(* Logix 5000 project; controller HP_SSC01hv vendor 1 type 14 code 158 rev 32.11; software revision 32.03; part 7 of 15 *)
(* tags used below, declared in another part *)
   A_C2_0422 : ALIAS FOR C2_Warning.22;
   A_C2_0423 : ALIAS FOR C2_Warning.23;
   A_C2_0425 : ALIAS FOR C2_Warning.25;
   A_C2_0426 : ALIAS FOR C2_Warning.26;
   C1_MAG : MOTION_INSTRUCTION;
   C1_MAS : MOTION_INSTRUCTION;
   C2_32HourTimers : TIMER[4];
   C2_ActualPositionMOD60 : REAL;
   C2_All_DLY_OK : BOOL;
   C2_Brake_Daily_ok : BOOL;
   C2_BrakeReleaseSelected : BOOL;
   C2_BrakeTestExpireTime : DINT;
   C2_BrakeTestExpireTimeTemp : DINT;
   C2_BrakeTestFailed : BOOL;
   C2_BrakeTestMessageNumber : DINT;
   C2_BrakeTestSelected : BOOL;
   C2_BrakeTestSequence : DINT;
   C2_BrakeTestWarning : BOOL;
   C2_DistanceToEvac : REAL;
   C2_Dump_OK : BOOL;
   C2_DumpValveReleaseSelected : BOOL;
   C2_DumpValveTestExpireTime : DINT;
   C2_DumpValveTestExpireTimeTemp : DINT;
   C2_DumpValveTestSelected : BOOL;
   C2_DumpValveTestSequence : DINT;
   C2_EvacPosition : REAL;
   C2_EvacPositionMOD60 : REAL;
   C2_ExcecutePBHoldTimer : TIMER;
   C2_FaultStandard : DINT;
   C2_GoNearOnPathDelay : TIMER;
   C2_GoToEvacMAM01 : MOTION_INSTRUCTION;
   C2_GoToOnPathMAM01 : MOTION_INSTRUCTION;
   C2_GoToOnPathMAM02 : MOTION_INSTRUCTION;
   C2_Home_OK : BOOL;
   C2_Homed : BOOL;
   C2_HomeExpireTime : DINT;
   C2_HomeExpireTimeTemp : DINT;
   C2_HomeSequence : DINT;
   C2_JogForwardFastSelected : BOOL;
   C2_JogForwardSlowSelected : BOOL;
   C2_JogReverseFastSelected : BOOL;
   C2_JogReverseSlowSelected : BOOL;
   C2_LubricationMessageNumber : DINT;
   C2_LubricationOnTimer : TIMER;
   C2_LubricationOverrideSelected : BOOL;
   C2_MAFR : MOTION_INSTRUCTION;
   C2_MAJDeceleration : REAL;
   C2_MASR : MOTION_INSTRUCTION;
   C2_Oiler : ALIAS FOR C2_RIO_AENT:O.Data[2].1;
   C2_OIT_BrakeRelease : BOOL;
   C2_OIT_BrakeReleaseDisplay : BOOL;
   C2_OIT_BrakeTest : BOOL;
   C2_OIT_BrakeTestDisplay : BOOL;
   C2_OIT_Command : DINT;
   C2_OIT_Current : DINT;
   C2_OIT_DumpValveRelease : BOOL;
   C2_OIT_DumpValveReleaseDisplay : BOOL;
   C2_OIT_DumpValveTest : BOOL;
   C2_OIT_DumpValveTestDisplay : BOOL;
   C2_OIT_FaultsExist : BOOL;
   C2_OIT_HomeCountDown : DINT;
   C2_OIT_JogForwardFast : BOOL;
   C2_OIT_JogForwardFastDisplay : BOOL;
   C2_OIT_JogForwardSlow : BOOL;
   C2_OIT_JogForwardSlowDisplay : BOOL;
   C2_OIT_JogReverseFast : BOOL;
   C2_OIT_JogReverseFastDisplay : BOOL;
   C2_OIT_JogReverseSlow : BOOL;
   C2_OIT_JogReverseSlowDisplay : BOOL;
   C2_OIT_JogStopDisplay : BOOL;
   C2_OIT_LubricationOverride : BOOL;
   C2_OIT_LubricationOverrideDisplay : BOOL;
   C2_OIT_PathError : DINT;
   C2_OIT_PathIndicatorHigh : DINT;
   C2_OIT_PathIndicatorLow : DINT;
   C2_OIT_WarningsExist : BOOL;
   C2_OneTryToFixErrorONS : BOOL;
   C2_ONS : DINT;
   C2_RemoteBrakeAndHomeSequence : DINT;
   C2_RemoteBrakeAndHomeSequenceAlarms : DINT;
   C2_RemoteBrakeAndHomeSequenceAlarmTimer : TIMER[8];
   C2_RemoteBrakeAndHomeSequenceONS : BOOL;
   C2_RemoteBrakeTestCMD : BOOL;
   C2_RemoteDumpTestCMD : BOOL;
   C2_RemoteHomeCMD : BOOL;
   C2_RemoteScreenMessageNumber : DINT;
   C2_RemoteSequenceDelay : TIMER[4];
   C2_RevolutionCounter : COUNTER;
   C2_ServoActionStatusOnDelay : TIMER;
   C2_TargetPositionError : REAL;
   C2_TargetPositionErrorTest : REAL;
   C2_Warning : DINT;
   MasterClockCopyMAS_Stop1 : MOTION_INSTRUCTION;
   MasterClockCopyMAS_Stop2 : MOTION_INSTRUCTION;
   MasterClockLocal : AXIS_VIRTUAL;
   none : BOOL;
   RCS_CMD_Auto_TON : TIMER;
   RCS_MasterClockLocalTagetDegrees : REAL;
   S_C2_FaultReset : BOOL;
   S_C2_FaultSafety : DINT;
   S_C2_ModeLocal : BOOL;
   S_C2_ModeRemote : BOOL;
   S_C2_MSTOP_InputOK : BOOL;
   S_C2_NearOnPath : BOOL;
   S_C2_NearOnPathHi : DINT;
   S_C2_NearOnPathLow : DINT;
   S_C2_OffPath : BOOL;
   S_C2_OnPath : BOOL;
   S_C2_PathError : DINT;
   S_RCS_MotionCMD_BrakeTest : BOOL;
   S_RCS_MotionCMD_Evac : BOOL;
   S_RCS_MotionCMD_GoNearOnPath : BOOL;
(* Carousel2, continued *)

ROUTINE C245_Lubrication   (* ladder *)
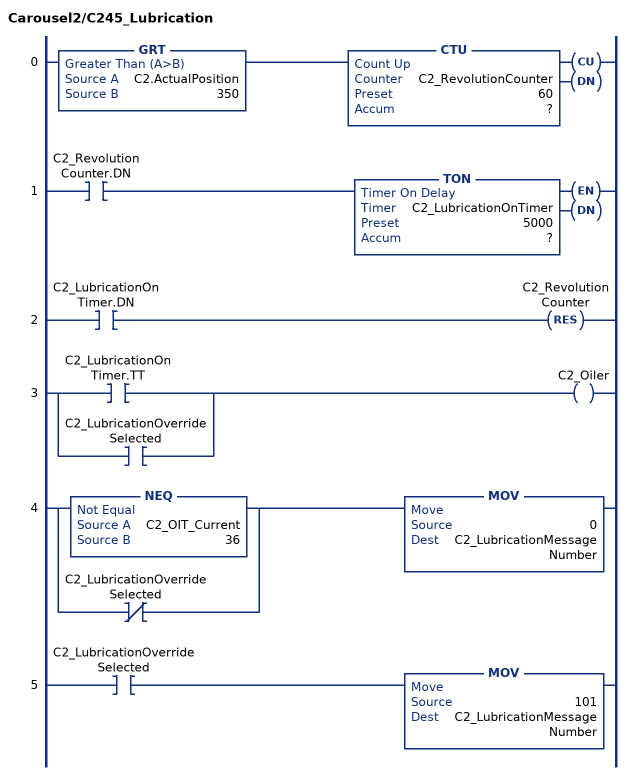
   0: GRT(C2.ActualPosition,350)CTU(C2_RevolutionCounter,?,?);
   1: XIC(C2_RevolutionCounter.DN)TON(C2_LubricationOnTimer,?,?);
   2: XIC(C2_LubricationOnTimer.DN)RES(C2_RevolutionCounter);
   3: [XIC(C2_LubricationOnTimer.TT) ,XIC(C2_LubricationOverrideSelected) ]OTE(C2_Oiler);
   4: [NEQ(C2_OIT_Current,36) ,XIO(C2_LubricationOverrideSelected) ]MOV(0,C2_LubricationMessageNumber);
   5: XIC(C2_LubricationOverrideSelected)MOV(101,C2_LubricationMessageNumber);
END_ROUTINE

ROUTINE C250_OIT   (* ladder *)
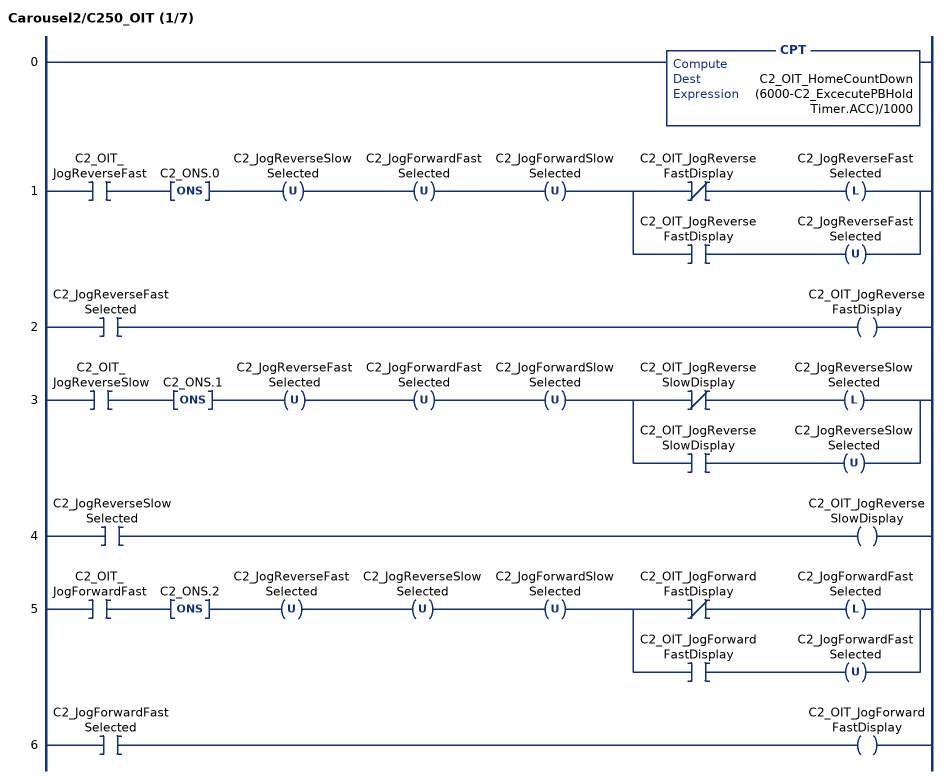
   0: CPT(C2_OIT_HomeCountDown,(6000-C2_ExcecutePBHoldTimer.ACC)/1000);
   1: XIC(C2_OIT_JogReverseFast)ONS(C2_ONS.0)OTU(C2_JogReverseSlowSelected)OTU(C2_JogForwardFastSelected)OTU(C2_JogForwardSlowSelected)[XIO(C2_OIT_JogReverseFastDisplay) OTL(C2_JogReverseFastSelected) ,XIC(C2_OIT_JogReverseFastDisplay) OTU(C2_JogReverseFastSelected) ];
   2: XIC(C2_JogReverseFastSelected)OTE(C2_OIT_JogReverseFastDisplay);
   3: XIC(C2_OIT_JogReverseSlow)ONS(C2_ONS.1)OTU(C2_JogReverseFastSelected)OTU(C2_JogForwardFastSelected)OTU(C2_JogForwardSlowSelected)[XIO(C2_OIT_JogReverseSlowDisplay) OTL(C2_JogReverseSlowSelected) ,XIC(C2_OIT_JogReverseSlowDisplay) OTU(C2_JogReverseSlowSelected) ];
   4: XIC(C2_JogReverseSlowSelected)OTE(C2_OIT_JogReverseSlowDisplay);
   5: XIC(C2_OIT_JogForwardFast)ONS(C2_ONS.2)OTU(C2_JogReverseFastSelected)OTU(C2_JogReverseSlowSelected)OTU(C2_JogForwardSlowSelected)[XIO(C2_OIT_JogForwardFastDisplay) OTL(C2_JogForwardFastSelected) ,XIC(C2_OIT_JogForwardFastDisplay) OTU(C2_JogForwardFastSelected) ];
   6: XIC(C2_JogForwardFastSelected)OTE(C2_OIT_JogForwardFastDisplay);
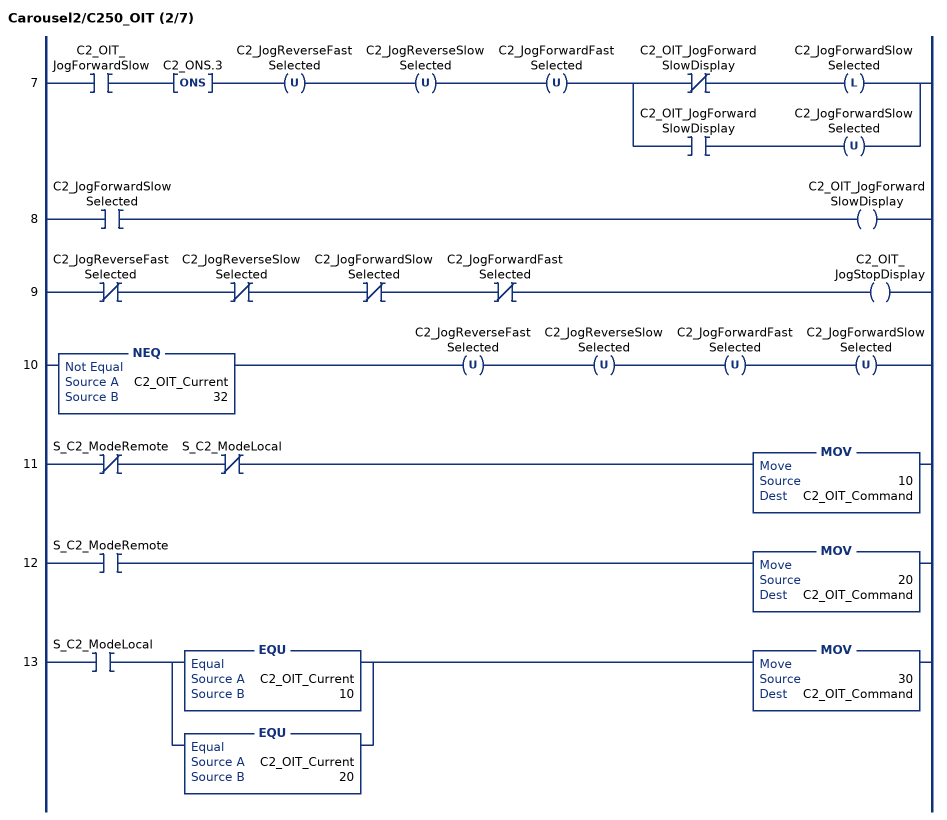
   7: XIC(C2_OIT_JogForwardSlow)ONS(C2_ONS.3)OTU(C2_JogReverseFastSelected)OTU(C2_JogReverseSlowSelected)OTU(C2_JogForwardFastSelected)[XIO(C2_OIT_JogForwardSlowDisplay) OTL(C2_JogForwardSlowSelected) ,XIC(C2_OIT_JogForwardSlowDisplay) OTU(C2_JogForwardSlowSelected) ];
   8: XIC(C2_JogForwardSlowSelected)OTE(C2_OIT_JogForwardSlowDisplay);
   9: XIO(C2_JogReverseFastSelected)XIO(C2_JogReverseSlowSelected)XIO(C2_JogForwardSlowSelected)XIO(C2_JogForwardFastSelected)OTE(C2_OIT_JogStopDisplay);
   10: NEQ(C2_OIT_Current,32)OTU(C2_JogReverseFastSelected)OTU(C2_JogReverseSlowSelected)OTU(C2_JogForwardFastSelected)OTU(C2_JogForwardSlowSelected);
   11: XIO(S_C2_ModeRemote)XIO(S_C2_ModeLocal)MOV(10,C2_OIT_Command);
   12: XIC(S_C2_ModeRemote)MOV(20,C2_OIT_Command);
   13: XIC(S_C2_ModeLocal)[EQU(C2_OIT_Current,10) ,EQU(C2_OIT_Current,20) ]MOV(30,C2_OIT_Command);
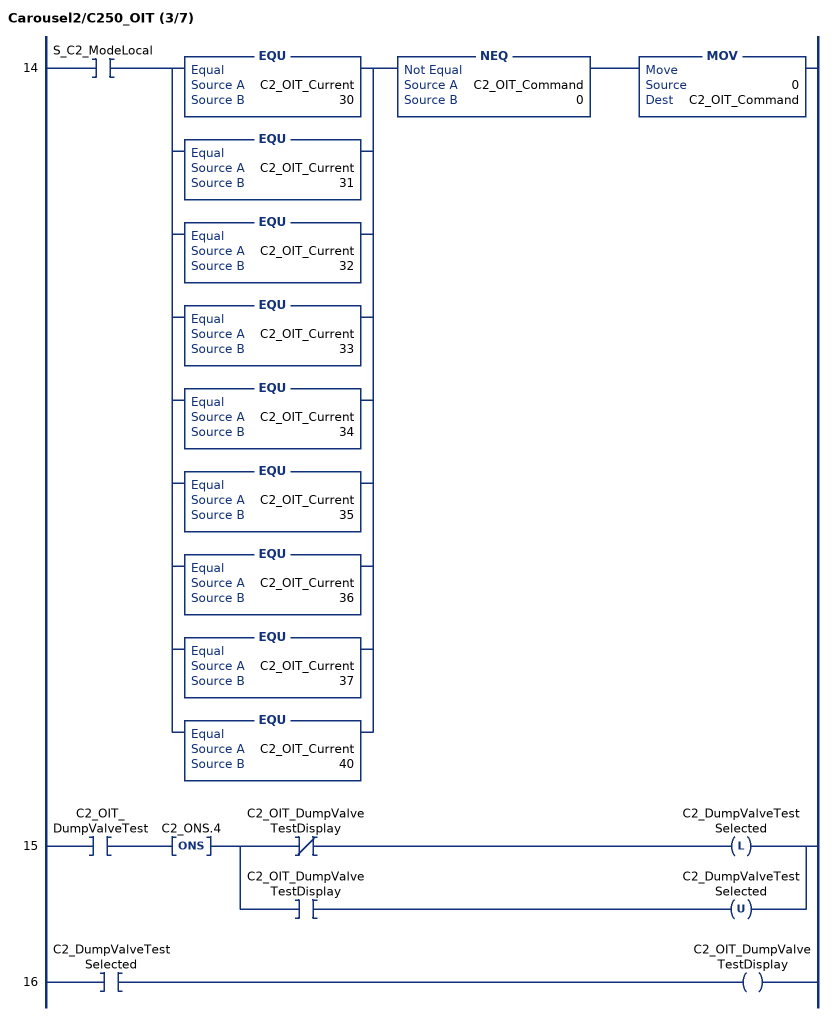
   14: XIC(S_C2_ModeLocal)[EQU(C2_OIT_Current,30) ,EQU(C2_OIT_Current,31) ,EQU(C2_OIT_Current,32) ,EQU(C2_OIT_Current,33) ,EQU(C2_OIT_Current,34) ,EQU(C2_OIT_Current,35) ,EQU(C2_OIT_Current,36) ,EQU(C2_OIT_Current,37) ,EQU(C2_OIT_Current,40) ]NEQ(C2_OIT_Command,0)MOV(0,C2_OIT_Command);
   15: XIC(C2_OIT_DumpValveTest)ONS(C2_ONS.4)[XIO(C2_OIT_DumpValveTestDisplay) OTL(C2_DumpValveTestSelected) ,XIC(C2_OIT_DumpValveTestDisplay) OTU(C2_DumpValveTestSelected) ];
   16: XIC(C2_DumpValveTestSelected)OTE(C2_OIT_DumpValveTestDisplay);
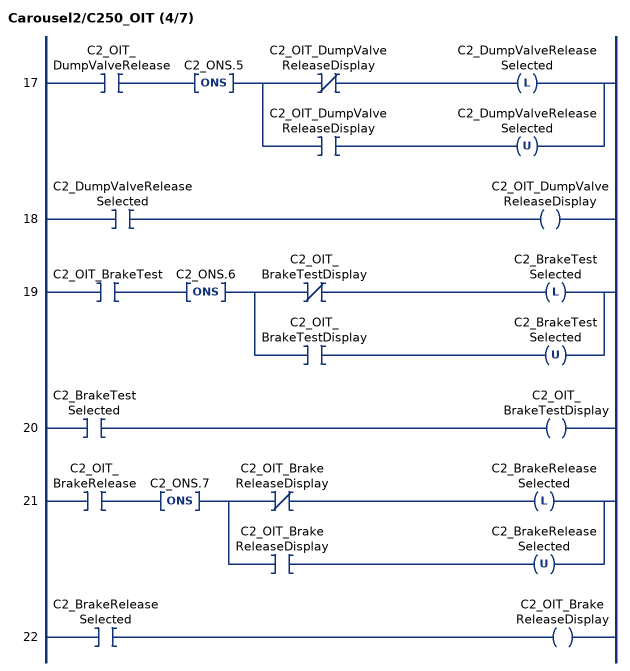
   17: XIC(C2_OIT_DumpValveRelease)ONS(C2_ONS.5)[XIO(C2_OIT_DumpValveReleaseDisplay) OTL(C2_DumpValveReleaseSelected) ,XIC(C2_OIT_DumpValveReleaseDisplay) OTU(C2_DumpValveReleaseSelected) ];
   18: XIC(C2_DumpValveReleaseSelected)OTE(C2_OIT_DumpValveReleaseDisplay);
   19: XIC(C2_OIT_BrakeTest)ONS(C2_ONS.6)[XIO(C2_OIT_BrakeTestDisplay) OTL(C2_BrakeTestSelected) ,XIC(C2_OIT_BrakeTestDisplay) OTU(C2_BrakeTestSelected) ];
   20: XIC(C2_BrakeTestSelected)OTE(C2_OIT_BrakeTestDisplay);
   21: XIC(C2_OIT_BrakeRelease)ONS(C2_ONS.7)[XIO(C2_OIT_BrakeReleaseDisplay) OTL(C2_BrakeReleaseSelected) ,XIC(C2_OIT_BrakeReleaseDisplay) OTU(C2_BrakeReleaseSelected) ];
   22: XIC(C2_BrakeReleaseSelected)OTE(C2_OIT_BrakeReleaseDisplay);
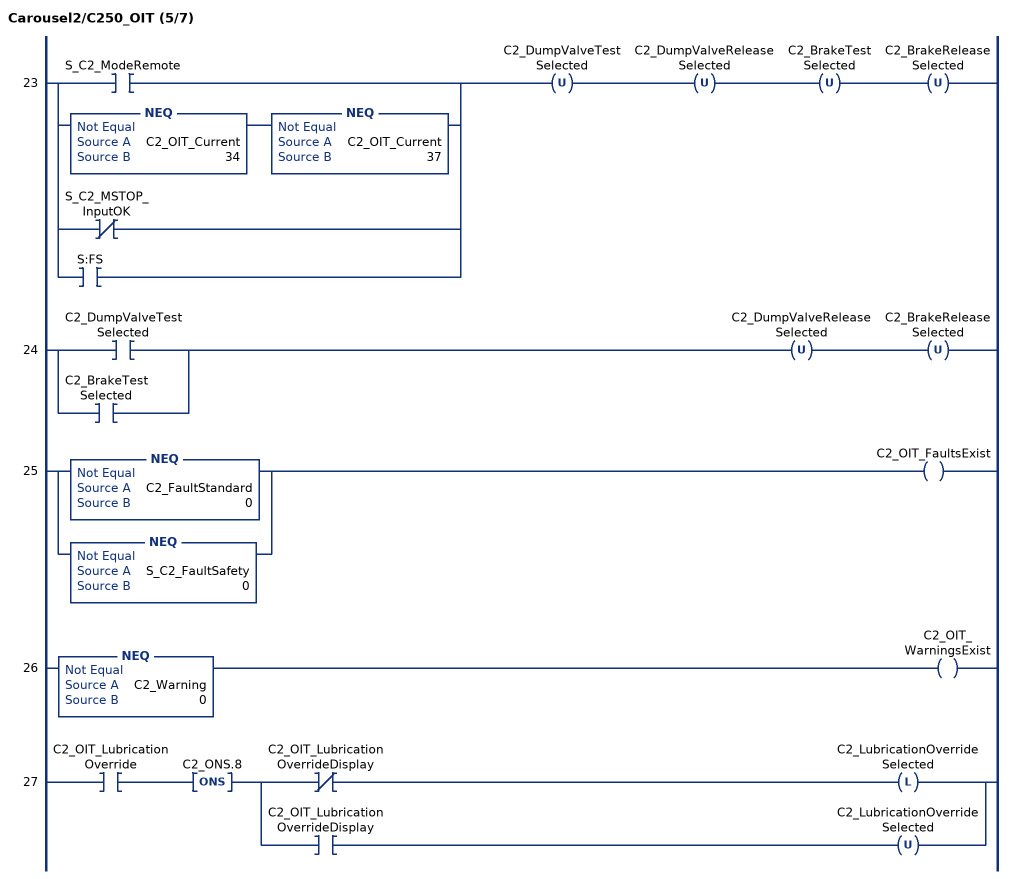
   23: [XIC(S_C2_ModeRemote) ,NEQ(C2_OIT_Current,34) NEQ(C2_OIT_Current,37) ,XIO(S_C2_MSTOP_InputOK) ,XIC(S:FS) ]OTU(C2_DumpValveTestSelected)OTU(C2_DumpValveReleaseSelected)OTU(C2_BrakeTestSelected)OTU(C2_BrakeReleaseSelected);
   24: [XIC(C2_DumpValveTestSelected) ,XIC(C2_BrakeTestSelected) ]OTU(C2_DumpValveReleaseSelected)OTU(C2_BrakeReleaseSelected);
   25: [NEQ(C2_FaultStandard,0) ,NEQ(S_C2_FaultSafety,0) ]OTE(C2_OIT_FaultsExist);
   26: NEQ(C2_Warning,0)OTE(C2_OIT_WarningsExist);
   27: XIC(C2_OIT_LubricationOverride)ONS(C2_ONS.8)[XIO(C2_OIT_LubricationOverrideDisplay) OTL(C2_LubricationOverrideSelected) ,XIC(C2_OIT_LubricationOverrideDisplay) OTU(C2_LubricationOverrideSelected) ];
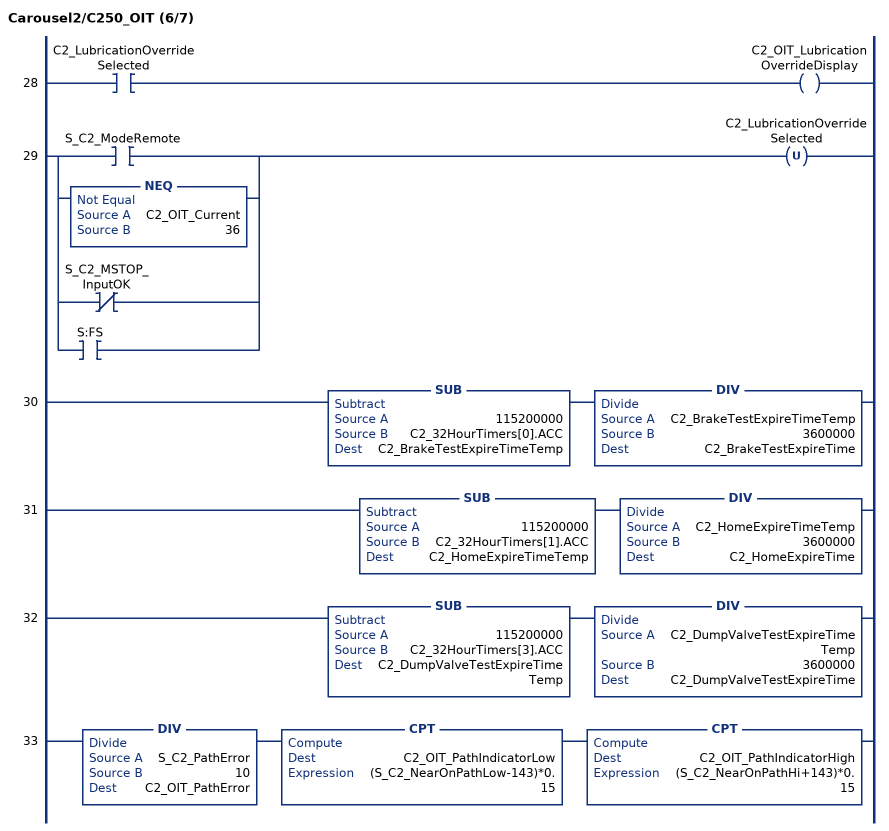
   28: XIC(C2_LubricationOverrideSelected)OTE(C2_OIT_LubricationOverrideDisplay);
   29: [XIC(S_C2_ModeRemote) ,NEQ(C2_OIT_Current,36) ,XIO(S_C2_MSTOP_InputOK) ,XIC(S:FS) ]OTU(C2_LubricationOverrideSelected);
   30: SUB(115200000,C2_32HourTimers[0].ACC,C2_BrakeTestExpireTimeTemp)DIV(C2_BrakeTestExpireTimeTemp,3600000,C2_BrakeTestExpireTime);
   31: SUB(115200000,C2_32HourTimers[1].ACC,C2_HomeExpireTimeTemp)DIV(C2_HomeExpireTimeTemp,3600000,C2_HomeExpireTime);
   32: SUB(115200000,C2_32HourTimers[3].ACC,C2_DumpValveTestExpireTimeTemp)DIV(C2_DumpValveTestExpireTimeTemp,3600000,C2_DumpValveTestExpireTime);
   33: DIV(S_C2_PathError,10,C2_OIT_PathError)CPT(C2_OIT_PathIndicatorLow,(S_C2_NearOnPathLow-143)*0.15)CPT(C2_OIT_PathIndicatorHigh,(S_C2_NearOnPathHi+143)*0.15);
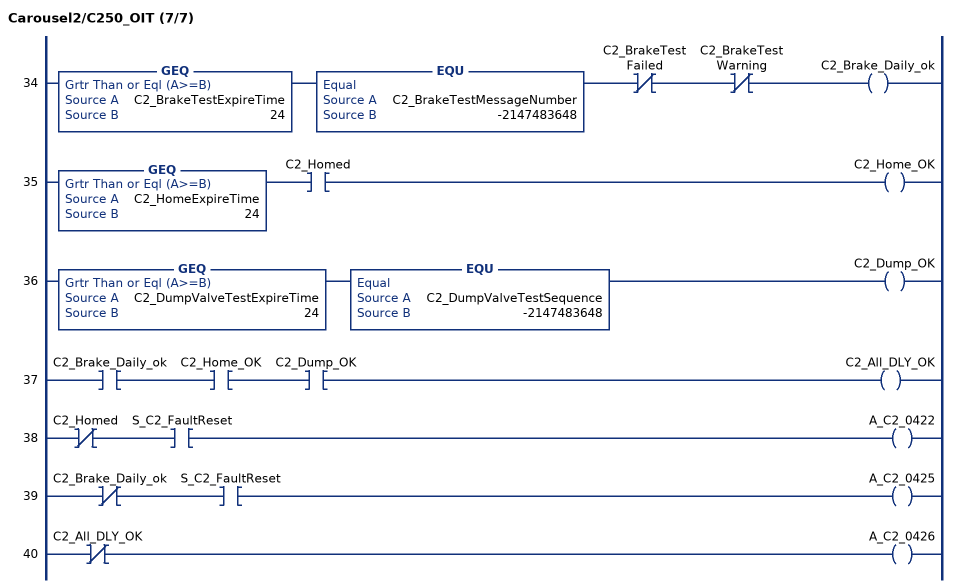
   34: GEQ(C2_BrakeTestExpireTime,24)EQU(C2_BrakeTestMessageNumber,-2147483648)XIO(C2_BrakeTestFailed)XIO(C2_BrakeTestWarning)OTE(C2_Brake_Daily_ok);
   35: GEQ(C2_HomeExpireTime,24)XIC(C2_Homed)OTE(C2_Home_OK);
   36: GEQ(C2_DumpValveTestExpireTime,24)EQU(C2_DumpValveTestSequence,-2147483648)OTE(C2_Dump_OK);
   37: XIC(C2_Brake_Daily_ok)XIC(C2_Home_OK)XIC(C2_Dump_OK)OTE(C2_All_DLY_OK);
   38: XIO(C2_Homed)XIC(S_C2_FaultReset)OTE(A_C2_0422);
   39: XIO(C2_Brake_Daily_ok)XIC(S_C2_FaultReset)OTE(A_C2_0425);
   40: XIO(C2_All_DLY_OK)OTE(A_C2_0426);
END_ROUTINE

ROUTINE C255_Remote   (* ladder *)
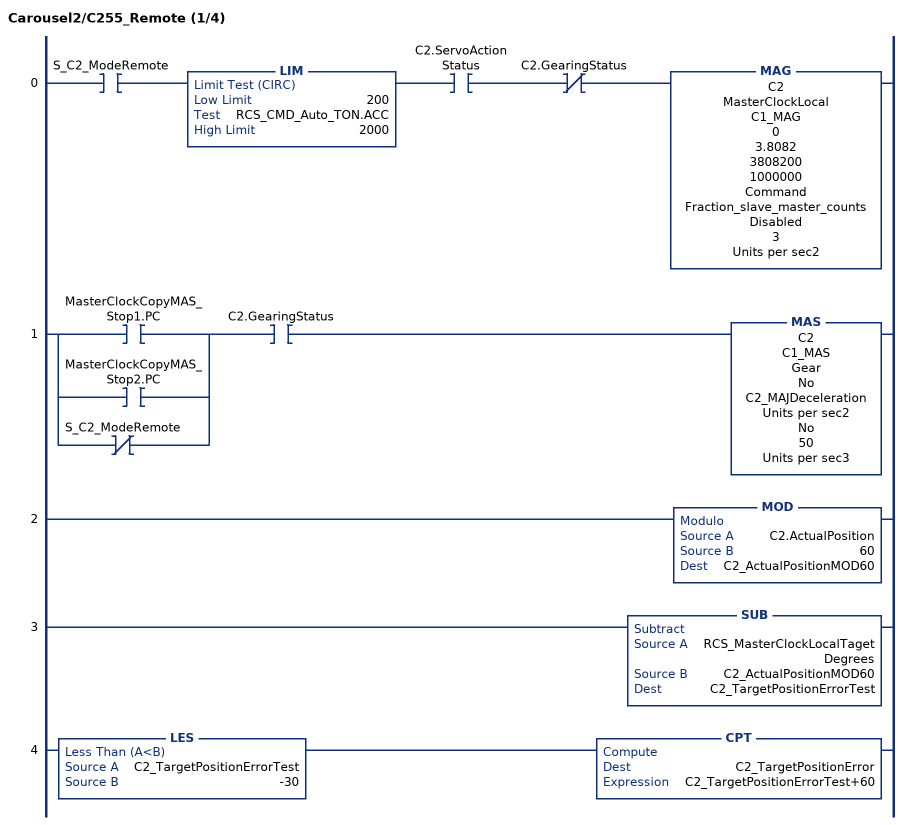
   0: XIC(S_C2_ModeRemote)LIM(200,RCS_CMD_Auto_TON.ACC,2000)XIC(C2.ServoActionStatus)XIO(C2.GearingStatus)MAG(C2,MasterClockLocal,C1_MAG,0,3.8082,3808200,1000000,Command,Fraction_slave_master_counts,Disabled,3,Units per sec2);
   1: [XIC(MasterClockCopyMAS_Stop1.PC) ,XIC(MasterClockCopyMAS_Stop2.PC) ,XIO(S_C2_ModeRemote) ]XIC(C2.GearingStatus)MAS(C2,C1_MAS,Gear,No,C2_MAJDeceleration,Units per sec2,No,50,Units per sec3);
   2: MOD(C2.ActualPosition,60,C2_ActualPositionMOD60);
   3: SUB(RCS_MasterClockLocalTagetDegrees,C2_ActualPositionMOD60,C2_TargetPositionErrorTest);
   4: LES(C2_TargetPositionErrorTest,-30)CPT(C2_TargetPositionError,C2_TargetPositionErrorTest+60);
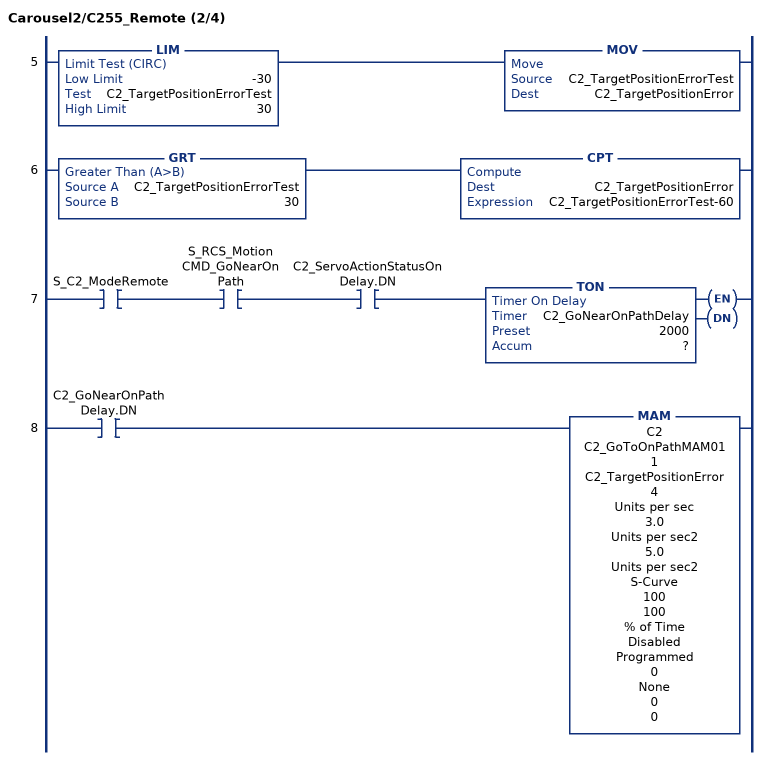
   5: LIM(-30,C2_TargetPositionErrorTest,30)MOV(C2_TargetPositionErrorTest,C2_TargetPositionError);
   6: GRT(C2_TargetPositionErrorTest,30)CPT(C2_TargetPositionError,C2_TargetPositionErrorTest-60);
   7: XIC(S_C2_ModeRemote)XIC(S_RCS_MotionCMD_GoNearOnPath)XIC(C2_ServoActionStatusOnDelay.DN)TON(C2_GoNearOnPathDelay,?,?);
   8: XIC(C2_GoNearOnPathDelay.DN)MAM(C2,C2_GoToOnPathMAM01,1,C2_TargetPositionError,4,Units per sec,3.0,Units per sec2,5.0,Units per sec2,S-Curve,100,100,% of Time,Disabled,Programmed,0,None,0,0);
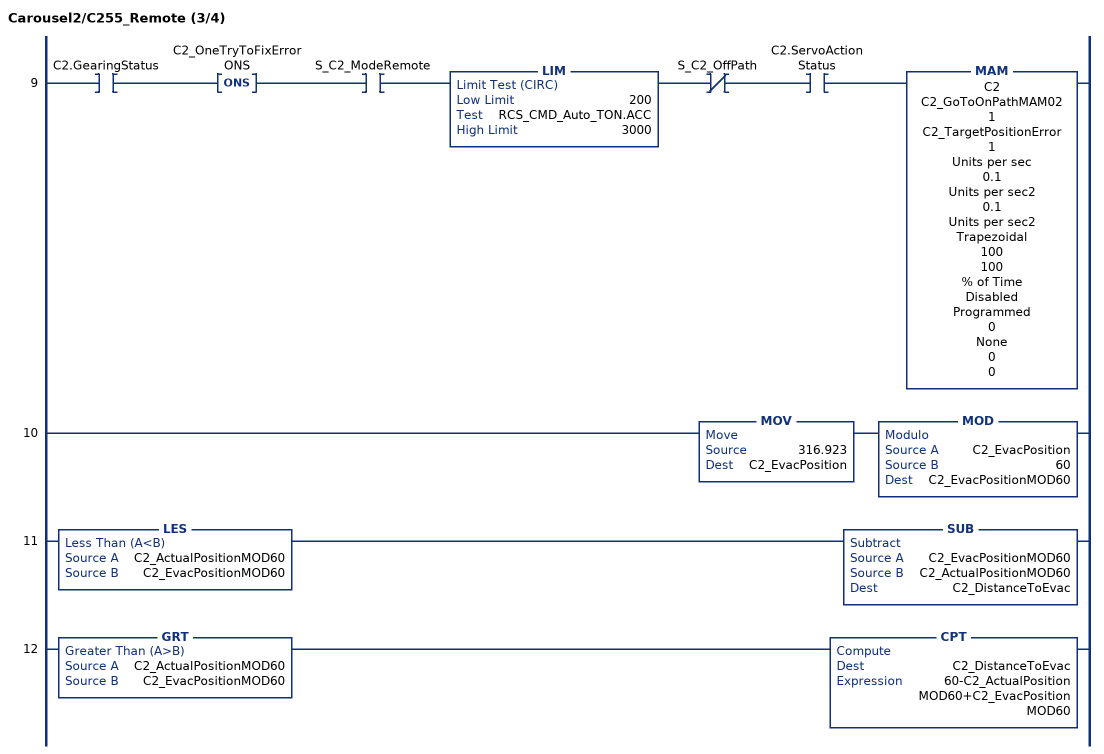
   9: XIC(C2.GearingStatus)ONS(C2_OneTryToFixErrorONS)XIC(S_C2_ModeRemote)LIM(200,RCS_CMD_Auto_TON.ACC,3000)XIO(S_C2_OffPath)XIC(C2.ServoActionStatus)MAM(C2,C2_GoToOnPathMAM02,1,C2_TargetPositionError,1,Units per sec,0.1,Units per sec2,0.1,Units per sec2,Trapezoidal,100,100,% of Time,Disabled,Programmed,0,None,0,0);
   10: MOV(316.923,C2_EvacPosition)MOD(C2_EvacPosition,60,C2_EvacPositionMOD60);
   11: LES(C2_ActualPositionMOD60,C2_EvacPositionMOD60)SUB(C2_EvacPositionMOD60,C2_ActualPositionMOD60,C2_DistanceToEvac);
   12: GRT(C2_ActualPositionMOD60,C2_EvacPositionMOD60)CPT(C2_DistanceToEvac,60-C2_ActualPositionMOD60+C2_EvacPositionMOD60);
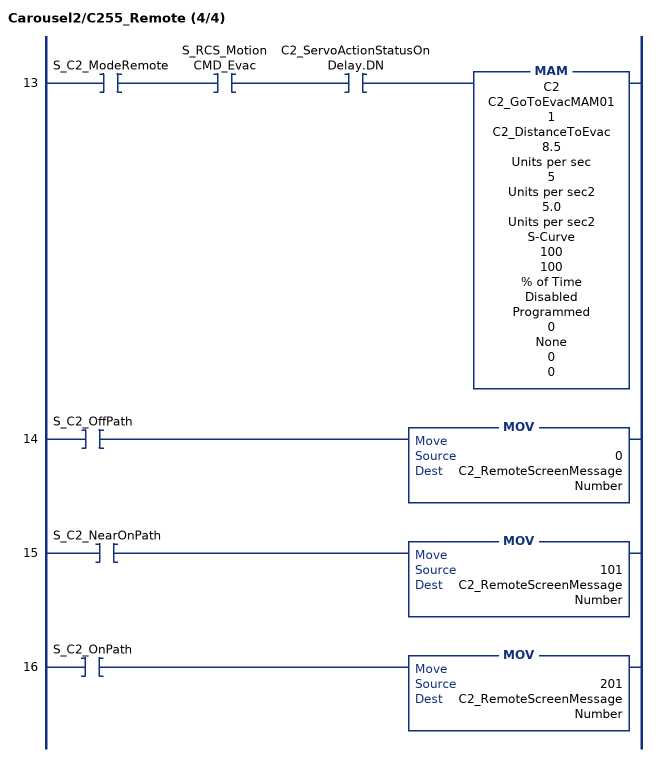
   13: XIC(S_C2_ModeRemote)XIC(S_RCS_MotionCMD_Evac)XIC(C2_ServoActionStatusOnDelay.DN)MAM(C2,C2_GoToEvacMAM01,1,C2_DistanceToEvac,8.5,Units per sec,5,Units per sec2,5.0,Units per sec2,S-Curve,100,100,% of Time,Disabled,Programmed,0,None,0,0);
   14: XIC(S_C2_OffPath)MOV(0,C2_RemoteScreenMessageNumber);
   15: XIC(S_C2_NearOnPath)MOV(101,C2_RemoteScreenMessageNumber);
   16: XIC(S_C2_OnPath)MOV(201,C2_RemoteScreenMessageNumber);
END_ROUTINE

ROUTINE C260_RemoteBrakeAndHome   (* ladder *)
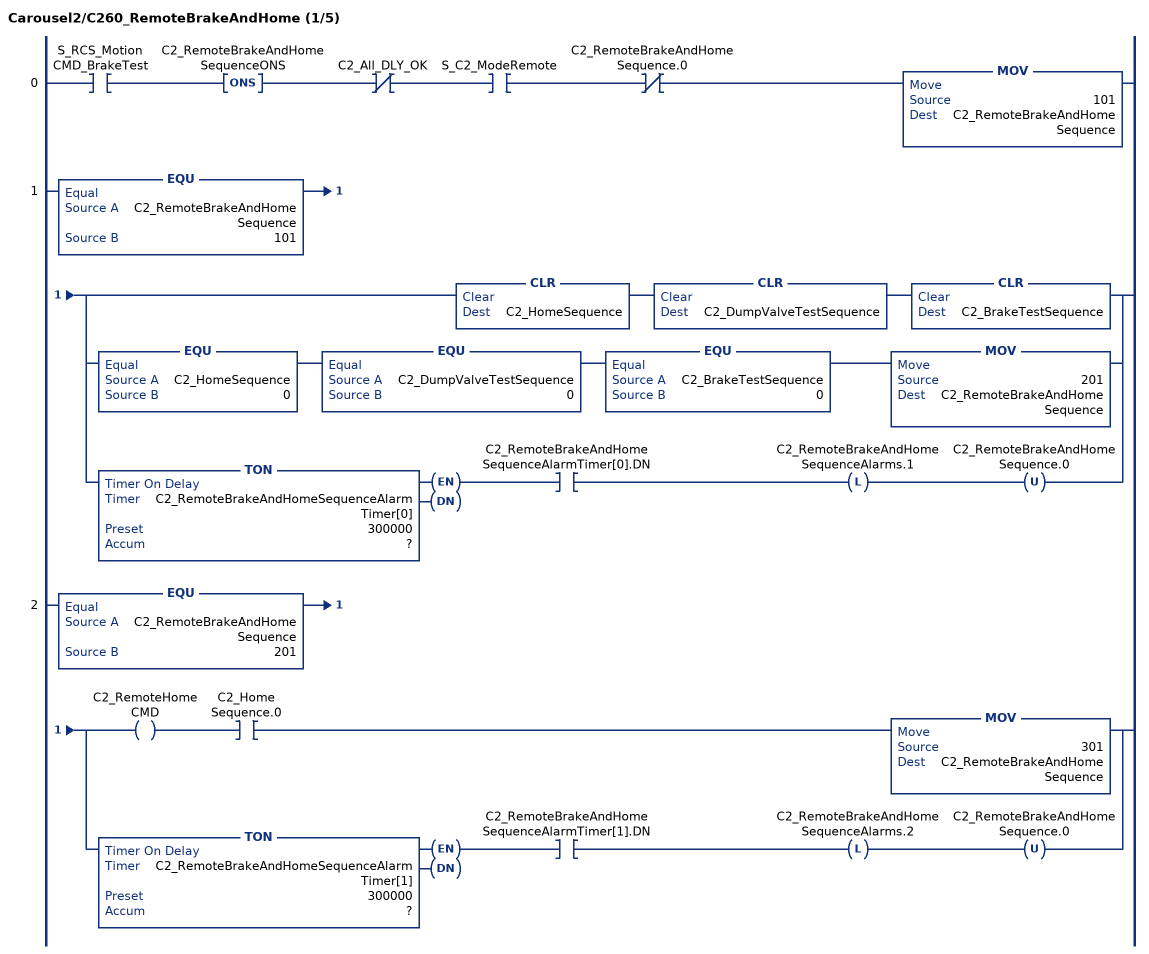
   0: XIC(S_RCS_MotionCMD_BrakeTest)ONS(C2_RemoteBrakeAndHomeSequenceONS)XIO(C2_All_DLY_OK)XIC(S_C2_ModeRemote)XIO(C2_RemoteBrakeAndHomeSequence.0)MOV(101,C2_RemoteBrakeAndHomeSequence);
   1: EQU(C2_RemoteBrakeAndHomeSequence,101)[CLR(C2_HomeSequence) CLR(C2_DumpValveTestSequence) CLR(C2_BrakeTestSequence) ,EQU(C2_HomeSequence,0) EQU(C2_DumpValveTestSequence,0) EQU(C2_BrakeTestSequence,0) MOV(201,C2_RemoteBrakeAndHomeSequence) ,TON(C2_RemoteBrakeAndHomeSequenceAlarmTimer[0],?,?) XIC(C2_RemoteBrakeAndHomeSequenceAlarmTimer[0].DN) OTL(C2_RemoteBrakeAndHomeSequenceAlarms.1) OTU(C2_RemoteBrakeAndHomeSequence.0) ];
   2: EQU(C2_RemoteBrakeAndHomeSequence,201)[OTE(C2_RemoteHomeCMD) XIC(C2_HomeSequence.0) MOV(301,C2_RemoteBrakeAndHomeSequence) ,TON(C2_RemoteBrakeAndHomeSequenceAlarmTimer[1],?,?) XIC(C2_RemoteBrakeAndHomeSequenceAlarmTimer[1].DN) OTL(C2_RemoteBrakeAndHomeSequenceAlarms.2) OTU(C2_RemoteBrakeAndHomeSequence.0) ];
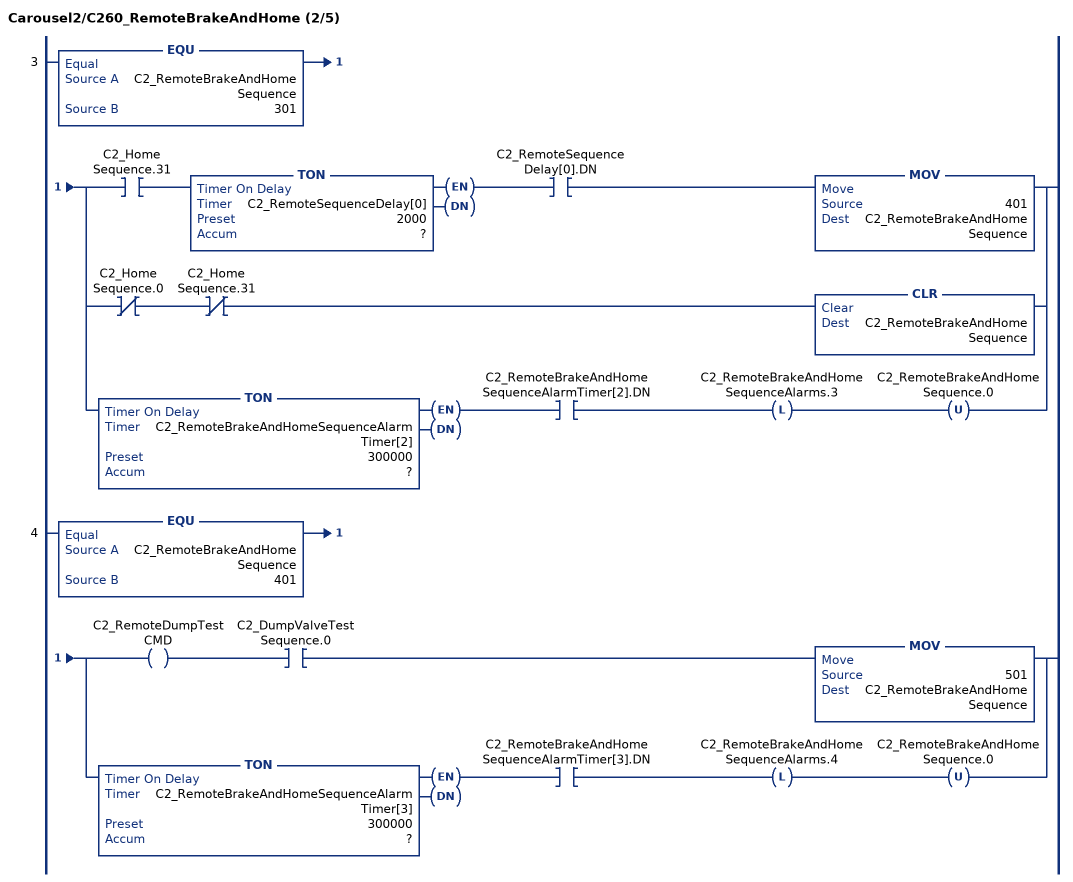
   3: EQU(C2_RemoteBrakeAndHomeSequence,301)[XIC(C2_HomeSequence.31) TON(C2_RemoteSequenceDelay[0],?,?) XIC(C2_RemoteSequenceDelay[0].DN) MOV(401,C2_RemoteBrakeAndHomeSequence) ,XIO(C2_HomeSequence.0) XIO(C2_HomeSequence.31) CLR(C2_RemoteBrakeAndHomeSequence) ,TON(C2_RemoteBrakeAndHomeSequenceAlarmTimer[2],?,?) XIC(C2_RemoteBrakeAndHomeSequenceAlarmTimer[2].DN) OTL(C2_RemoteBrakeAndHomeSequenceAlarms.3) OTU(C2_RemoteBrakeAndHomeSequence.0) ];
   4: EQU(C2_RemoteBrakeAndHomeSequence,401)[OTE(C2_RemoteDumpTestCMD) XIC(C2_DumpValveTestSequence.0) MOV(501,C2_RemoteBrakeAndHomeSequence) ,TON(C2_RemoteBrakeAndHomeSequenceAlarmTimer[3],?,?) XIC(C2_RemoteBrakeAndHomeSequenceAlarmTimer[3].DN) OTL(C2_RemoteBrakeAndHomeSequenceAlarms.4) OTU(C2_RemoteBrakeAndHomeSequence.0) ];
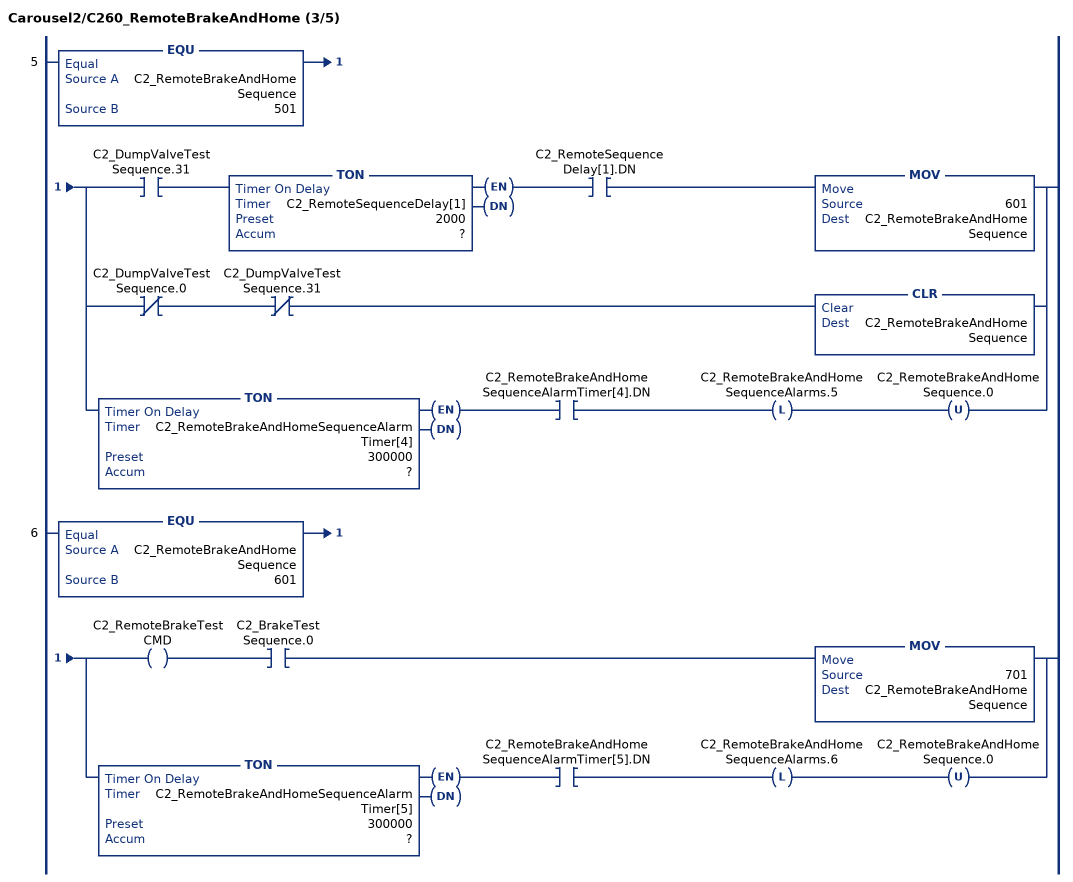
   5: EQU(C2_RemoteBrakeAndHomeSequence,501)[XIC(C2_DumpValveTestSequence.31) TON(C2_RemoteSequenceDelay[1],?,?) XIC(C2_RemoteSequenceDelay[1].DN) MOV(601,C2_RemoteBrakeAndHomeSequence) ,XIO(C2_DumpValveTestSequence.0) XIO(C2_DumpValveTestSequence.31) CLR(C2_RemoteBrakeAndHomeSequence) ,TON(C2_RemoteBrakeAndHomeSequenceAlarmTimer[4],?,?) XIC(C2_RemoteBrakeAndHomeSequenceAlarmTimer[4].DN) OTL(C2_RemoteBrakeAndHomeSequenceAlarms.5) OTU(C2_RemoteBrakeAndHomeSequence.0) ];
   6: EQU(C2_RemoteBrakeAndHomeSequence,601)[OTE(C2_RemoteBrakeTestCMD) XIC(C2_BrakeTestSequence.0) MOV(701,C2_RemoteBrakeAndHomeSequence) ,TON(C2_RemoteBrakeAndHomeSequenceAlarmTimer[5],?,?) XIC(C2_RemoteBrakeAndHomeSequenceAlarmTimer[5].DN) OTL(C2_RemoteBrakeAndHomeSequenceAlarms.6) OTU(C2_RemoteBrakeAndHomeSequence.0) ];
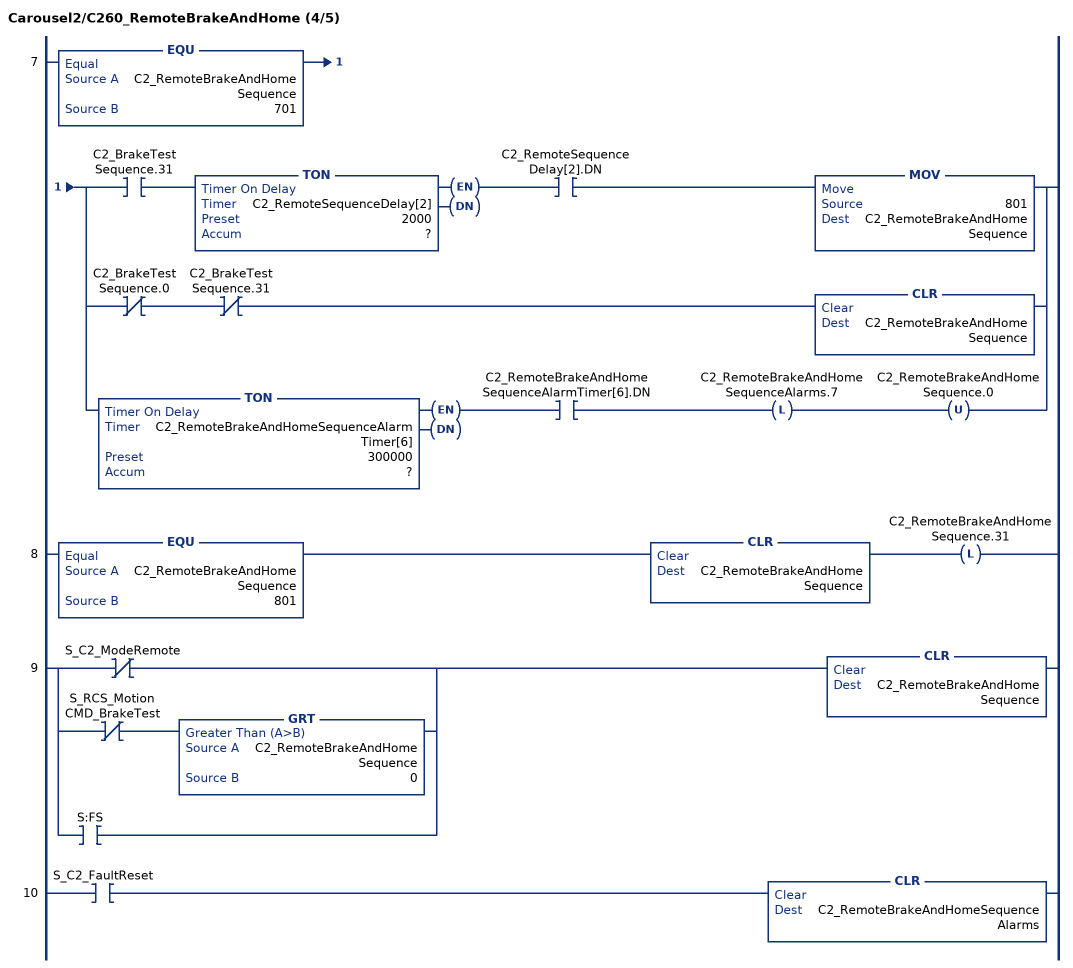
   7: EQU(C2_RemoteBrakeAndHomeSequence,701)[XIC(C2_BrakeTestSequence.31) TON(C2_RemoteSequenceDelay[2],?,?) XIC(C2_RemoteSequenceDelay[2].DN) MOV(801,C2_RemoteBrakeAndHomeSequence) ,XIO(C2_BrakeTestSequence.0) XIO(C2_BrakeTestSequence.31) CLR(C2_RemoteBrakeAndHomeSequence) ,TON(C2_RemoteBrakeAndHomeSequenceAlarmTimer[6],?,?) XIC(C2_RemoteBrakeAndHomeSequenceAlarmTimer[6].DN) OTL(C2_RemoteBrakeAndHomeSequenceAlarms.7) OTU(C2_RemoteBrakeAndHomeSequence.0) ];
   8: EQU(C2_RemoteBrakeAndHomeSequence,801)CLR(C2_RemoteBrakeAndHomeSequence)OTL(C2_RemoteBrakeAndHomeSequence.31);
   9: [XIO(S_C2_ModeRemote) ,XIO(S_RCS_MotionCMD_BrakeTest) GRT(C2_RemoteBrakeAndHomeSequence,0) ,XIC(S:FS) ]CLR(C2_RemoteBrakeAndHomeSequence);
   10: XIC(S_C2_FaultReset)CLR(C2_RemoteBrakeAndHomeSequenceAlarms);
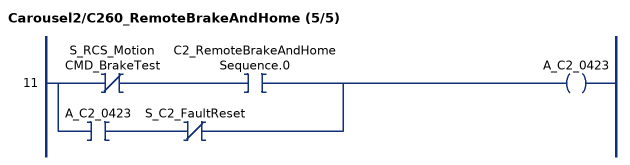
   11: [XIO(S_RCS_MotionCMD_BrakeTest) XIC(C2_RemoteBrakeAndHomeSequence.0) ,XIC(A_C2_0423) XIO(S_C2_FaultReset) ]OTE(A_C2_0423);
END_ROUTINE

ROUTINE C265_Reset   (* ladder *)
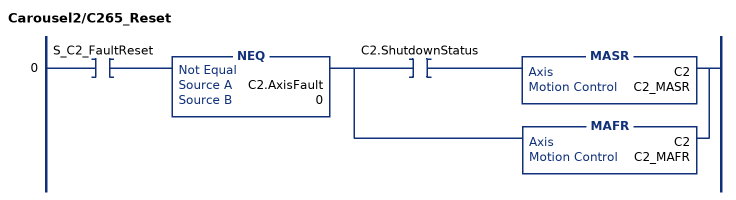
   0: XIC(S_C2_FaultReset)NEQ(C2.AxisFault,0)[XIC(C2.ShutdownStatus) MASR(C2,C2_MASR) ,MAFR(C2,C2_MAFR) ];
END_ROUTINE
END_PROGRAM
